FUNCTION_BLOCK DosagemAlcalinizante (* Composite Function Block Type *)
  (* Standard: 61499-2 *)
  (* Version 0.0, 02/03/2026, template *)
  PACKAGE Hidryco.HidrycoLib;
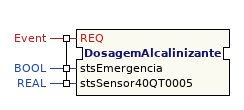
  EVENT_INPUT
    REQ WITH stsSensor40QT0005, stsEmergencia;
  END_EVENT
  VAR_INPUT
    stsEmergencia : BOOL;
    stsSensor40QT0005 : REAL;
  END_VAR
  (* 0 - INITIALIZATION *)
  (* 1 - FUNCTIONAL INPUT INTERFACE *)
  (* 6 - OT-IT INTERFACE *)
  (* 2 - FUNCTIONAL OUTPUT INTERFACE *)
  (* 3 - FIELD INTERFACE *)
  (* 4 - CHILDREN *)
  (* 5 - LOGICS *)
  (* 5.B - OPERATION MODE MANAGEMENT *)
  (* 5.C - INTERLOCKS MANAGEMENT *)
  (* 5.A - FUNCTIONAL BEHAVIORS *)
  FBS
    BO_800_02 : Motor_Partida_Direta;
    DO_800_04 : Motor_Dosagem;
    DO_800_05 : Motor_Dosagem;
    LIT_800_03 : Sensor_Nivel_4a20;
    Revezamento : Revezamento_3_Motores(stsDisponivelEquipamento3 := FALSE);
    comandoAutomatico1 : comandoAutomatico(stsDisponivelEquipamento3 := FALSE, stsNecessidadeHabilitado := FALSE);
    plcStart1 : plcStart(Prio := 10);
    IThis : DosagemAlcalinizante_HMI(QI := TRUE);
    PID : PID;
    comandoAutomatico2 : comandoAutomatico(stsRevezamentoHabilitado := FALSE, stsNecessidadeHabilitado := FALSE, stsDisponivelEquipamento2 := FALSE, stsDisponivelEquipamento3 := FALSE);
    Bloq_800_04 : BloqueioAtivaDesativa;
    Bloq_800_05 : BloqueioAtivaDesativa;
  END_FBS
  EVENT_CONNECTIONS
    Revezamento.E_ATUALIZA_HABILITADO TO comandoAutomatico1.E_ATUALIZA_HABILITADOS;
    Revezamento.E_ATUALIZA_EQUIPAMENTO_PRINCIPAL TO comandoAutomatico1.E_ATUALIZA_EQUIPAMENTO_PRINCIPAL;
    DO_800_05.CNF TO Revezamento.E_ATUALIZA_DISPONIBILIDADE_EQUIPAMENTO;
    DO_800_04.CNF TO Revezamento.E_ATUALIZA_DISPONIBILIDADE_EQUIPAMENTO;
    DO_800_04.CNF TO comandoAutomatico1.E_ATUALIZA_DISPONIBILIDADE_EQUIPAMENTOS;
    DO_800_05.CNF TO comandoAutomatico1.E_ATUALIZA_DISPONIBILIDADE_EQUIPAMENTOS;
    REQ TO PID.E_ATUALIZA_PV;
    BO_800_02.CNF TO comandoAutomatico2.E_ATUALIZA_DISPONIBILIDADE_EQUIPAMENTOS;
    BO_800_02.CNF TO comandoAutomatico2.E_ATUALIZA_HABILITADOS;
    LIT_800_03.E_AUALIZA_SENSOR_HABILITADO TO Bloq_800_04.E_ATUALIZA_SENSOR;
    LIT_800_03.E_ATUALIZA_SENSOR TO Bloq_800_04.E_ATUALIZA_SENSOR;
    LIT_800_03.E_AUALIZA_SENSOR_HABILITADO TO Bloq_800_05.E_ATUALIZA_SENSOR;
    LIT_800_03.E_ATUALIZA_SENSOR TO Bloq_800_05.E_ATUALIZA_SENSOR;
    plcStart1.FIRST_INIT TO IThis.AB8817508E95161;
    plcStart1.REDO_INIT TO IThis.AB8817508E95161;
    IThis.3E9DCB3F6C290B63 TO BO_800_02.E_RESET_FALHAS;
    IThis.3E9DCB3F6C290B63 TO DO_800_04.E_RESET_FALHAS;
    IThis.3E9DCB3F6C290B63 TO DO_800_05.E_RESET_FALHAS;
    REQ TO BO_800_02.REQ;
    REQ TO DO_800_04.REQ;
    REQ TO DO_800_05.REQ;
    comandoAutomatico2.E_ATUALIZA_COMANDO_AUTOMATICO TO BO_800_02.REQ;
    Bloq_800_04.E_ATUALIZA_BLOQUEIO TO BO_800_02.REQ;
    Bloq_800_05.E_ATUALIZA_BLOQUEIO TO DO_800_04.REQ;
    Bloq_800_05.E_ATUALIZA_BLOQUEIO TO DO_800_05.REQ;
    comandoAutomatico1.E_ATUALIZA_COMANDO_AUTOMATICO TO DO_800_05.REQ;
    comandoAutomatico1.E_ATUALIZA_COMANDO_AUTOMATICO TO DO_800_04.REQ;
    PID.E_ATUALIZA_SAIDA TO DO_800_04.REQ;
    PID.E_ATUALIZA_SAIDA TO DO_800_05.REQ;
    PID.E_ATUALIZA_PID_HABILITADO TO DO_800_04.REQ;
    PID.E_ATUALIZA_PID_HABILITADO TO DO_800_05.REQ;
    IThis.89BF3FE22E96B211 TO plcStart1.ACK_FIRST;
  END_CONNECTIONS
  DATA_CONNECTIONS
    Revezamento.stsRevezamentoHabilitado TO comandoAutomatico1.stsRevezamentoHabilitado;
    Revezamento.stsEquipamentoPrincipal TO comandoAutomatico1.stsEquipamentoPrincipal;
    DO_800_04.stsDisponivelAutomatico TO Revezamento.stsDisponivelEquipamento1;
    DO_800_05.stsDisponivelAutomatico TO Revezamento.stsDisponivelEquipamento2;
    DO_800_04.stsDisponivelAutomatico TO comandoAutomatico1.stsDisponivelEquipamento1;
    DO_800_05.stsDisponivelAutomatico TO comandoAutomatico1.stsDisponivelEquipamento2;
    comandoAutomatico1.cmdAutomaticoEquipamento1 TO DO_800_04.cmdLigarAutomatico;
    comandoAutomatico1.cmdAutomaticoEquipamento2 TO DO_800_05.cmdLigarAutomatico;
    stsSensor40QT0005 TO PID.stsPv;
    PID.stsPIDHabilitado TO DO_800_04.stsPIDHabilitado;
    PID.stsPIDHabilitado TO DO_800_05.stsPIDHabilitado;
    PID.stsSaida TO DO_800_04.stsSaidaAutomatico;
    PID.stsSaida TO DO_800_05.stsSaidaAutomatico;
    BO_800_02.stsDiponivelAutomatico TO comandoAutomatico2.stsDisponivelEquipamento1;
    Bloq_800_04.stsBloqueioAutomatico TO BO_800_02.bloqueioAutomatico;
    LIT_800_03.stsSensorHabilitado TO Bloq_800_04.stsSensorHabilitado;
    LIT_800_03.stsSensor TO Bloq_800_04.stsSensor;
    LIT_800_03.stsFalhaSensor TO Bloq_800_04.stsFalhaSensor;
    LIT_800_03.stsSensorHabilitado TO Bloq_800_05.stsSensorHabilitado;
    LIT_800_03.stsSensor TO Bloq_800_05.stsSensor;
    LIT_800_03.stsFalhaSensor TO Bloq_800_05.stsFalhaSensor;
    Bloq_800_05.stsBloqueioAutomatico TO DO_800_05.stsBloqueioAutomatico;
    Bloq_800_05.stsBloqueioAutomatico TO DO_800_04.stsBloqueioAutomatico;
    IThis.3F76E9CCEE1C62DE TO BO_800_02.cmdResetFalhas;
    IThis.3F76E9CCEE1C62DE TO DO_800_04.cmdResetFalhas;
    IThis.3F76E9CCEE1C62DE TO DO_800_05.cmdResetFalhas;
    stsEmergencia TO BO_800_02.CF68B7C2C7F473D9;
    stsEmergencia TO DO_800_04.5C85E7B3BE347ADB;
    stsEmergencia TO DO_800_05.5C85E7B3BE347ADB;
  END_CONNECTIONS
END_FUNCTION_BLOCK
